FUNCTION F_FehlerAufgetreten : BOOL
(* Soll eine Fehlerauswertung gemacht werden oer nicht *)
VAR_INPUT
END_VAR
VAR
	akku : DWORD;
END_VAR

(* Netzwerk: 6 *** Fehler aufgetreten ? *)

(*
L MD 100
L MD 104
OD -- ODER-Doppelwort
L MD 108
OD -- ODER-Doppelwort
L 0
<>D -- 	AKKU2 ungleich AKKU1 [DWORD], also wenn die Merker Fehler enthalten...ist VKE 1
= "M0.7" M0.7 -- Störung aufgetreten (gesammelt)
*)
GVL.errsAsDword := F_GetErrorsAsDWORD(errStruct := GVL.errs);
//...größerer Umbau gegenüber altem AWL-Programm, aber vom Prinzip her gleich.
VAT.bSammelStoerung := GVL.errsAsDword <> 0; //Sammel-Störung

(*
SPB X027 -- Springe wenn VKE = 1, ... zu X027, also überspringe RETURN.
BEA -- Bausteinende absolut, im Falle KEINES Fehlers: Keine Fehlerbitauswertung
*)
IF NOT VAT.bSammelStoerung THEN
	F_FehlerAufgetreten := FALSE;
	RETURN;
END_IF

//...jetzt noch nachsehen, ob SAFETY ok ist...
(*
X027: UN "T 72" T72 -- Verz. Alles OK von SAFETY (früher PNOZ), Fage ist SAFETY FALSE ?
BEB -- Bausteinende bedingt, Wenn SAFETY auch FALSE: auch Keine Fehlerbitauswertung 
*)

IF NOT GVL.tonSAFETYok.Q THEN
	F_FehlerAufgetreten := FALSE; //Wenn SAFETY = FALSE, Keine Fehlerbitauswertung 
	RETURN;
END_IF

F_FehlerAufgetreten := TRUE; //Auswertung fahren...

END_FUNCTION

(* stored: Version 1.1.0.1, ProductVersion 3.1.4024.3
   POU F_FehlerAufgetreten: Id {bcaff27b-2f82-4c7a-b883-1308bf1a5a7e}, SpecialFunc None *)
